{attribute 'qualified_only'}
{attribute 'strict'}
{attribute 'to_string'}
TYPE eRobPosType :
(
	Absolut := 0,			// Absolute Bewegung bezogen auf Basis-Koordinatensystem
	Relativ := 1			// Relative Bewegung bezogen auf aktuelle Position
);
END_TYPE

(* stored: Version 1.1.0.1
   DUT eRobPosType: Id {1c3dc3d5-5f39-4411-b92b-135ff03411c6} *)
